TYPE ST_KeyenceLaser_Count_Result_Data :
STRUCT
END_STRUCT
END_TYPE

(* stored: Version 1.1.0.1, ProductVersion 3.1.4024.11
   DUT ST_KeyenceLaser_Count_Result_Data: Id {0c67ccf7-d206-4b0b-a803-10128af0dfdd} *)
